// TIA Portal V20 export
DATA_BLOCK "R_Parameters"   // DB124
{ S7_Optimized_Access := 'TRUE' }
// stored: MemoryReserve 100
   VAR
      "$R[96]" { S7_SetPoint := 'True'} : SINU_typeNcVarTokenLReal;
      "$R[97]" { S7_SetPoint := 'True'} : SINU_typeNcVarTokenLReal;
      "$R[95]" { S7_SetPoint := 'True'} : SINU_typeNcVarTokenLReal;
      "$R[94]" { S7_SetPoint := 'True'} : SINU_typeNcVarTokenLReal;
   END_VAR
BEGIN
   "$R[96]".token.syntaxId := 16#82;
   "$R[96]".token.areaAndUnit := 16#41;
   "$R[96]".token.column := 16#1;
   "$R[96]".token.row := 16#61;
   "$R[96]".token.blockType := 16#15;
   "$R[96]".token.rowCount := 16#1;
   "$R[96]".token.dataType := 16#F;
   "$R[96]".token.length := 16#8;
   "$R[97]".token.syntaxId := 16#82;
   "$R[97]".token.areaAndUnit := 16#41;
   "$R[97]".token.column := 16#1;
   "$R[97]".token.row := 16#62;
   "$R[97]".token.blockType := 16#15;
   "$R[97]".token.rowCount := 16#1;
   "$R[97]".token.dataType := 16#F;
   "$R[97]".token.length := 16#8;
   "$R[95]".token.syntaxId := 16#82;
   "$R[95]".token.areaAndUnit := 16#41;
   "$R[95]".token.column := 16#1;
   "$R[95]".token.row := 16#60;
   "$R[95]".token.blockType := 16#15;
   "$R[95]".token.rowCount := 16#1;
   "$R[95]".token.dataType := 16#F;
   "$R[95]".token.length := 16#8;
   "$R[94]".token.syntaxId := 16#82;
   "$R[94]".token.areaAndUnit := 16#41;
   "$R[94]".token.column := 16#1;
   "$R[94]".token.row := 16#5F;
   "$R[94]".token.blockType := 16#15;
   "$R[94]".token.rowCount := 16#1;
   "$R[94]".token.dataType := 16#F;
   "$R[94]".token.length := 16#8;
END_DATA_BLOCK
